FUNCTION_BLOCK SP_Dispensing (* Dispensing parameters (none): OPC UA IDs, range check and latching *)
  (* Standard: 61499-2 *)
  (* Version 0.1, 2026-09-28, Project contributors, AAU Smart Production Lab *)
  PACKAGE filling;
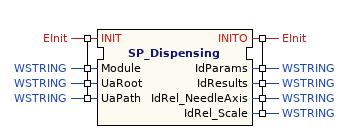
  EVENT_INPUT
    INIT : EInit WITH Module, UaRoot, UaPath;
  END_EVENT
  EVENT_OUTPUT
    INITO : EInit WITH IdParams, IdResults, IdRel_NeedleAxis, IdRel_Scale;
  END_EVENT
  VAR_INPUT
    Module : WSTRING;
    UaRoot : WSTRING;
    UaPath : WSTRING;
  END_VAR
  VAR_OUTPUT
    IdParams : WSTRING;
    IdResults : WSTRING;
    IdRel_NeedleAxis : WSTRING;
    IdRel_Scale : WSTRING;
  END_VAR
  EC_STATES
    INIT : INIT -> INITO;
  END_STATES
  ALGORITHM INIT IN ST:
IdParams := "";
IdResults := CONCAT(CONCAT(CONCAT("opc_ua[WRITE;", CONCAT(UaRoot, UaPath)), "/Results/Weight"), "]");
IdRel_NeedleAxis := CONCAT(CONCAT("loc[", Module), "/NeedleAxis/cmd]");
IdRel_Scale := CONCAT(CONCAT("loc[", Module), "/Scale/cmd]");
  END_ALGORITHM
END_FUNCTION_BLOCK
